(* IEC 61131-3 sources: AXOpen/src/showcase/app/src/core/AXOpen.Messaging, 3 files *)

(* ---- AxoIncidentBarExample.st ---- *)
USING AXOpen.Core;
USING AXOpen.Messaging;
USING AXOpen.Messaging.Static;

NAMESPACE AxoIncidentBarExample

    // Demonstrates AxoCauseAnalyzer + AxoIncidentBarView with a nested twin-tree topology.
    // Operator toggles condition BOOLs to fire Error/Critical messengers at multiple
    // tree levels. The bar ranks the upper messenger as 'top cause' because it
    // owns more downstream alarms (Symbol-prefix heuristic) and shares the burst window.
    {S7.extern=ReadWrite}
    CLASS IncidentTopology EXTENDS AXOpen.Core.AxoObject
        //<TopologyDeclaration>
        VAR PUBLIC
            {#ix-set:AttributeName = "<#Station (top of the topology)#>"}
            station : Station;
        END_VAR
        //</TopologyDeclaration>

        VAR PRIVATE
            _rootObject : AxoObject;
        END_VAR

        METHOD PUBLIC Execute
            _rootObject.Run(THIS);
            station.Run(_rootObject);
        END_METHOD
    END_CLASS

    {S7.extern=ReadWrite}
    CLASS PUBLIC Station EXTENDS AXOpen.Core.AxoObject
        //<StationDeclaration>
        VAR PUBLIC
            {#ix-set:AttributeName = "<#Station-level alarm (Error)#>"}
            {#ix-set:PlcTextList = "[1]:'<#Station emergency stop active#>':'<#Station has tripped the safety chain. Resolve all downstream issues before resetting.#>'"}
            _station_messenger : AXOpen.Messaging.Static.AxoMessenger;
            {#ix-set:AttributeName = "<#Trigger Station error#>"}
            _station_error : BOOL;

            {#ix-attr:[Container(Layout.Stack)]}
            drive : Drive;

            {#ix-attr:[Container(Layout.Stack)]}
            conveyor : Conveyor;
        END_VAR
        //</StationDeclaration>

        METHOD PUBLIC OVERRIDE Run
            VAR_INPUT
                inParent : IAxoObject;
            END_VAR
            SUPER.Run(inParent);
            _station_messenger.Serve(THIS);
            //<StationActivate>
            _station_messenger.ActivateOnCondition(ULINT#1, _station_error, eAxoMessageCategory#Error)
                              .RequireAcknowledgement();
            //</StationActivate>
            drive.Run(THIS);
            conveyor.Run(THIS);
        END_METHOD
    END_CLASS

    {S7.extern=ReadWrite}
    CLASS PUBLIC Drive EXTENDS AXOpen.Core.AxoObject
        //<DriveDeclaration>
        VAR PUBLIC
            {#ix-set:AttributeName = "<#Drive over-current (Critical)#>"}
            {#ix-set:PlcTextList = "[1]:'<#Drive over-current trip#>':'<#Inverter detected current above the safety limit. Check load and wiring.#>'"}
            _drive_messenger : AXOpen.Messaging.Static.AxoMessenger;
            {#ix-set:AttributeName = "<#Trigger Drive over-current#>"}
            _drive_error : BOOL;

            {#ix-attr:[Container(Layout.Stack)]}
            encoder : Encoder;
        END_VAR
        //</DriveDeclaration>

        METHOD PUBLIC OVERRIDE Run
            VAR_INPUT
                inParent : IAxoObject;
            END_VAR
            SUPER.Run(inParent);
            _drive_messenger.Serve(THIS);
            _drive_messenger.ActivateOnCondition(ULINT#1, _drive_error, eAxoMessageCategory#Critical)
                            .RequireAcknowledgement();
            encoder.Run(THIS);
        END_METHOD
    END_CLASS

    {S7.extern=ReadWrite}
    CLASS PUBLIC Encoder EXTENDS AXOpen.Core.AxoObject
        VAR PUBLIC
            {#ix-set:AttributeName = "<#Encoder signal lost (Error)#>"}
            {#ix-set:PlcTextList = "[1]:'<#Encoder signal lost#>':'<#The drive lost feedback from the encoder. Check cable continuity and connector seating.#>'"}
            _encoder_messenger : AXOpen.Messaging.Static.AxoMessenger;
            {#ix-set:AttributeName = "<#Trigger Encoder signal lost#>"}
            _encoder_error : BOOL;
        END_VAR

        METHOD PUBLIC OVERRIDE Run
            VAR_INPUT
                inParent : IAxoObject;
            END_VAR
            SUPER.Run(inParent);
            _encoder_messenger.Serve(THIS);
            _encoder_messenger.ActivateOnCondition(ULINT#1, _encoder_error, eAxoMessageCategory#Error)
                              .RequireAcknowledgement();
        END_METHOD
    END_CLASS

    {S7.extern=ReadWrite}
    CLASS PUBLIC Conveyor EXTENDS AXOpen.Core.AxoObject
        VAR PUBLIC
            {#ix-set:AttributeName = "<#Conveyor jammed (Error)#>"}
            {#ix-set:PlcTextList = "[1]:'<#Conveyor jammed#>':'<#Detected motor stall while pulley still commanded. Clear the obstruction and reset.#>'"}
            _conveyor_messenger : AXOpen.Messaging.Static.AxoMessenger;
            {#ix-set:AttributeName = "<#Trigger Conveyor jam#>"}
            _conveyor_error : BOOL;

            {#ix-attr:[Container(Layout.Stack)]}
            sensor : Sensor;
        END_VAR

        METHOD PUBLIC OVERRIDE Run
            VAR_INPUT
                inParent : IAxoObject;
            END_VAR
            SUPER.Run(inParent);
            _conveyor_messenger.Serve(THIS);
            _conveyor_messenger.ActivateOnCondition(ULINT#1, _conveyor_error, eAxoMessageCategory#Error)
                               .RequireAcknowledgement();
            sensor.Run(THIS);
        END_METHOD
    END_CLASS

    {S7.extern=ReadWrite}
    CLASS PUBLIC Sensor EXTENDS AXOpen.Core.AxoObject
        VAR PUBLIC
            {#ix-set:AttributeName = "<#Sensor disconnected (Error)#>"}
            {#ix-set:PlcTextList = "[1]:'<#Sensor disconnected#>':'<#Photo-eye lost present feedback. Verify alignment and 24V supply.#>'"}
            _sensor_messenger : AXOpen.Messaging.Static.AxoMessenger;
            {#ix-set:AttributeName = "<#Trigger Sensor disconnect#>"}
            _sensor_error : BOOL;
        END_VAR

        METHOD PUBLIC OVERRIDE Run
            VAR_INPUT
                inParent : IAxoObject;
            END_VAR
            SUPER.Run(inParent);
            _sensor_messenger.Serve(THIS);
            _sensor_messenger.ActivateOnCondition(ULINT#1, _sensor_error, eAxoMessageCategory#Error)
                             .RequireAcknowledgement();
        END_METHOD
    END_CLASS

END_NAMESPACE

(* ---- AxoStaticMessengerDocuExample.st ---- *)
USING AXOpen.Messaging;
USING AXOpen.Messaging.Static;

NAMESPACE AxoStaticMessengerDocuExample
    {S7.extern=ReadWrite}
    CLASS MessengersExamples EXTENDS AXOpen.Core.AxoObject
        VAR PUBLIC
            {#ix-set:AttributeName = "<#Messenger 1 - activate using 'Activate' method called inside the if statement#>"}
            {#ix-set:PlcTextList = "[1]:'<#Messenger 1: message text for message code 1#>':'<#Messenger 1: help text for message code 1#>';[2]:'<#Messenger 1: message text for message code 2#>':'<#Messenger 1: help text for message code 2#>';[3]:'<#Messenger 1: message text for message code 3#>':'<#Messenger 1: help text for message code 3#>';[4]:'<#Messenger 1: message text for message code 4#>':'<#Messenger 1: help text for message code 4#>';[5]:'<#Messenger 1: message text for message code 5#>':'<#Messenger 1: help text for message code 5#>';[6]:'<#Messenger 1: message text for message code 6#>':'<#Messenger 1: help text for message code 6#>';[7]:'<#Messenger 1: message text for message code 7#>':'<#Messenger 1: help text for message code 7#>';[8]:'<#Messenger 1: message text for message code 8#>':'<#Messenger 1: help text for message code 8#>';[9]:'<#Messenger 1: message text for message code 9#>':'<#Messenger 1: help text for message code 9#>';[10]:'<#Messenger 1: message text for message code 10#>':'<#Messenger 1: help text for message code 10#>';[11]:'<#Messenger 1: message text for message code 11#>':'<#Messenger 1: help text for message code 11#>'"}
            _messenger1 : AXOpen.Messaging.Static.AxoMessenger;
            {#ix-attr:[Container(Layout.Wrap)]}
            {#ix-set:AttributeName = "<#Set to high to activate the messenger 1#>"}
            _messenger1condition : BOOL;
            {#ix-set:AttributeName = "<#message 1 code#>"}
            _messenger1code : UINT;

            {#ix-attr:[Container(Layout.Stack)]}
            {#ix-set:AttributeName = "<#Messenger 2 - activate using 'ActivateOnCondition' method called cyclically#>"}
            {#ix-set:PlcTextList = "[1]:'<#Messenger 2: message text for message code 1#>':'<#Messenger 2: help text for message code 1#>'[2]:'<#Messenger 2: message text for message code 2#>':'<#Messenger 2: help text for message code 2#>'"}
            _messenger2 : AXOpen.Messaging.Static.AxoMessenger;
            {#ix-attr:[Container(Layout.Wrap)]}
            {#ix-set:AttributeName = "<#Set to high to activate the messenger 2#>"}
            _messenger2condition : BOOL;
            {#ix-set:AttributeName = "<#message 2 code#>"}
            _messenger2code : UINT;

            {#ix-attr:[Container(Layout.Stack)]}
            {#ix-set:AttributeName = "<#Messenger 3 - one message example, long help text#>"}
            {#ix-set:PlcTextList = "[1]:'<#Message text for messenger 3#>':'<#Lorem ipsum dolor sit amet, consectetur adipiscing elit. Phasellus neque eros, malesuada ac orci ut, ornare ullamcorper purus. Integer ultrices turpis vel est suscipit blandit. Mauris blandit eros augue, in mollis dui tincidunt vel. Sed placerat augue risus, eget pulvinar felis dictum quis. Aliquam ut interdum nisl. Aliquam et velit id turpis blandit laoreet nec ut ligula. Aliquam ac neque risus. Fusce porta mauris eget nulla iaculis mattis. Etiam auctor mi eget libero laoreet, sed interdum ipsum pellentesque. Maecenas vitae quam vitae velit tincidunt fringilla. Fusce sagittis elit sit amet tempor pretium. Donec elementum, ligula at laoreet mollis, est ipsum elementum lectus, et mollis nisi tellus id erat. In hac habitasse platea dictumst.#>'"}
            _messenger3 : AXOpen.Messaging.Static.AxoMessenger;
            {#ix-set:AttributeName = "<#Set to high to activate the messenger 3#>"}
            _messenger3condition : BOOL;

            {#ix-attr:[Container(Layout.Stack)]}
            //<PlcTextListDeclaration>
            {#ix-set:AttributeName = "<#Messenger 4 - textlist in PLC#>"}
            {#ix-set:PlcTextList = "[1]:'<#Messenger 4: static message text for message code 1 declared in the PLC code#>':'<#Messenger 4: static help text for message code 1 declared in the PLC code#>'[2]:'<#Messenger 4: static message text for message code 2 declared in the PLC code#>':'<#Messenger 4: static help text for message code 2 declared in the PLC code#>'"}
            _messenger4 : AXOpen.Messaging.Static.AxoMessenger;
            //</PlcTextListDeclaration>
            {#ix-set:AttributeName = "<#Set to high to activate the messenger 4 with message code 1#>"}
            _messenger4condition_1 : BOOL;
            {#ix-set:AttributeName = "<#Set to high to activate the messenger 4 with message code 2#>"}
            _messenger4condition_2 : BOOL;

            {#ix-attr:[Container(Layout.Stack)]}
            //<TextListGoingToBeDeclaredInDotNet>
            {#ix-set:AttributeName = "<#Messenger 5 - textlist in .NET#>"}
            _messenger5 : AXOpen.Messaging.Static.AxoMessenger;
            //</TextListGoingToBeDeclaredInDotNet>
            {#ix-attr:[Container(Layout.Wrap)]}
            {#ix-set:AttributeName = "<#Set to high to activate the messenger 5 with code 1#>"}
            _messenger5condition_1 : BOOL;
            {#ix-set:AttributeName = "<#Set to high to activate the messenger 5 with code 2#>"}
            _messenger5condition_2 : BOOL;
            {#ix-set:AttributeName = "<#Set to high to activate the messenger 5 with code 3#>"}
            _messenger5condition_3 : BOOL;
            {#ix-set:AttributeName = "<#Set to high to activate the messenger 5 with code 4#>"}
            _messenger5condition_4 : BOOL;
            {#ix-set:AttributeName = "<#Set to high to activate the messenger 5 with code 5#>"}
            _messenger5condition_5 : BOOL;
            {#ix-set:AttributeName = "<#Set to high to activate the messenger 5 with code 6#>"}
            _messenger5condition_6 : BOOL;
            {#ix-set:AttributeName = "<#Set to high to activate the messenger 5 with code 7#>"}
            _messenger5condition_7 : BOOL;
            {#ix-set:AttributeName = "<#Set to high to activate the messenger 5 with code 8#>"}
            _messenger5condition_8 : BOOL;
            {#ix-set:AttributeName = "<#Set to high to activate the messenger 5 with code 9#>"}
            _messenger5condition_9 : BOOL;
            {#ix-set:AttributeName = "<#Set to high to activate the messenger 5 with code 10, with no help text defined#>"}
            _messenger5condition_10 : BOOL;
            {#ix-set:AttributeName = "<#Set to high to call the messenger 5#>"}
            _messenger5callcondition : BOOL;

            {#ix-attr:[Container(Layout.Stack)]}
            {#ix-set:AttributeName = "<#Messenger 6 - invalid implementation#>"}
            {#ix-set:PlcTextList = "[1]:'<#Messenger 6: static message text for message code 1 declared in the PLC code#>':'<#Messenger 6: static help text for message code 1 declared in the PLC code#>'[2]:'<#Messenger 6: static message text for message code 2 declared in the PLC code#>':'<#Messenger 6: static help text for message code 2 declared in the PLC code#>'"}
            _messenger6 : AXOpen.Messaging.Static.AxoMessenger;
            {#ix-set:AttributeName = "<#Set to high to activate the messenger 6 with message code 1#>"}
            _messenger6condition_1 : BOOL;
            {#ix-set:AttributeName = "<#Set to high to activate the messenger 6 with message code 2#>"}
            _messenger6condition_2 : BOOL;
        END_VAR

        VAR PRIVATE
            _rootObject :   AxoObject;
        END_VAR
        METHOD PUBLIC Execute
            _rootObject.Run(THIS);
            //<Activate>
            _messenger1.Serve(_rootObject);
            IF _messenger1condition THEN
                _messenger1.Activate(_messenger1code,eAxoMessageCategory#Error);
            END_IF;
            //</Activate>

            //<ActivateOnCondition>
            _messenger2.Serve(_rootObject);
            _messenger2.ActivateOnCondition(_messenger2code,_messenger2condition,eAxoMessageCategory#Warning).RequireAcknowledgement();
            //</ActivateOnCondition>

            //<RequireAcknowledgement>
            _messenger2.Serve(_rootObject);
            _messenger2.ActivateOnCondition(_messenger2code,_messenger2condition,eAxoMessageCategory#Warning).RequireAcknowledgement();
            //</RequireAcknowledgement>

            //<DoNotRequireAcknowledgement>
            _messenger3.Serve(_rootObject);
            _messenger3.ActivateOnCondition(UINT#1,_messenger3condition,eAxoMessageCategory#Error).DoNotRequireAcknowledgement();
            //</DoNotRequireAcknowledgement>

            //<ActivateOnConditionWithMessageCodeTextListDeclaredInThePlcCode>
            _messenger4.Serve(_rootObject);
            _messenger4.ActivateOnCondition(UINT#1,_messenger4condition_1,eAxoMessageCategory#Info).RequireAcknowledgement();
            _messenger4.ActivateOnCondition(UINT#2,_messenger4condition_2,eAxoMessageCategory#Info).RequireAcknowledgement();
            //</ActivateOnConditionWithMessageCodeTextListDeclaredInThePlcCode>

            //<ActivateOnConditionWithMessageCodeTextListDeclaredInDotNet>
            IF _messenger5callcondition THEN
                _messenger5.Serve(_rootObject);
                _messenger5.ActivateOnCondition(ULINT#1,_messenger5condition_1,eAxoMessageCategory#Error).RequireAcknowledgement();
                _messenger5.ActivateOnCondition(ULINT#2,_messenger5condition_2,eAxoMessageCategory#Error).RequireAcknowledgement();
                _messenger5.ActivateOnCondition(ULINT#3,_messenger5condition_3,eAxoMessageCategory#Error).RequireAcknowledgement();
                _messenger5.ActivateOnCondition(ULINT#4,_messenger5condition_4,eAxoMessageCategory#Error).RequireAcknowledgement();
                _messenger5.ActivateOnCondition(ULINT#5,_messenger5condition_5,eAxoMessageCategory#Error).RequireAcknowledgement();
                _messenger5.ActivateOnCondition(ULINT#6,_messenger5condition_6,eAxoMessageCategory#Error).RequireAcknowledgement();
                _messenger5.ActivateOnCondition(ULINT#7,_messenger5condition_7,eAxoMessageCategory#Error).RequireAcknowledgement();
                _messenger5.ActivateOnCondition(ULINT#8,_messenger5condition_8,eAxoMessageCategory#Error).RequireAcknowledgement();
                _messenger5.ActivateOnCondition(ULINT#9,_messenger5condition_9,eAxoMessageCategory#Error).RequireAcknowledgement();
                _messenger5.ActivateOnCondition(ULINT#10,_messenger5condition_10,eAxoMessageCategory#Error).RequireAcknowledgement();
            ELSE
                _messenger5.Restore();
            END_IF;
            //</ActivateOnConditionWithMessageCodeTextListDeclaredInDotNet>

            //<InvalidImplementation>
            _messenger6.ActivateOnCondition(UINT#1,_messenger6condition_1,eAxoMessageCategory#Info).RequireAcknowledgement();
            _messenger6.ActivateOnCondition(UINT#2,_messenger6condition_2,eAxoMessageCategory#Info).RequireAcknowledgement();
            _messenger6.Serve(_rootObject);
            //</InvalidImplementation>
        END_METHOD
    END_CLASS

    //<MessengerCompleteExample
    {S7.extern=ReadWrite}
    CLASS Messengers EXTENDS AXOpen.Core.AxoObject
        VAR PUBLIC
            {#ix-set:PlcTextList = "[10]:'<#Messenger 1: static message text for message code 10 declared in the PLC code#>':'<#Messenger 1: static help text for message code 10 declared in the PLC code#>'"}
            _messenger1 : AXOpen.Messaging.Static.AxoMessenger;
            {#ix-set:AttributeName = "<#Set to high to activate the messenger 1#>"}
            _messenger1condition : BOOL;

            {#ix-set:PlcTextList = "[10]:'<#Messenger 2: static message text for message code 10 declared in the PLC code#>':'<#Messenger 2: static help text for message code 10 declared in the PLC code#>'"}
            _messenger2 : AXOpen.Messaging.Static.AxoMessenger;
            {#ix-set:AttributeName = "<#Set to high to activate the messenger 2#>"}
            _messenger2condition : BOOL;

            {#ix-set:PlcTextList = "[10]:'<#Messenger 3: static message text for message code 10 declared in the PLC code#>':'<#Messenger 3: static help text for message code 10 declared in the PLC code#>';[20]:'<#Messenger 3: static message text for message code 20 declared in the PLC code#>':'<#Messenger 3: static help text for message code 20 declared in the PLC code#>'"}
            _messenger3 : AXOpen.Messaging.Static.AxoMessenger;
            {#ix-set:AttributeName = "<#Set to high to activate the messenger 3 with message code 10#>"}
            _messenger3condition_10 : BOOL;
            {#ix-set:AttributeName = "<#Set to high to activate the messenger 3 with message code 20#>"}
            _messenger3condition_20 : BOOL;

            _messenger4 : AXOpen.Messaging.Static.AxoMessenger;
            {#ix-set:AttributeName = "<#Set to high to activate the messenger 4 with message code 10#>"}
            _messenger4condition_10 : BOOL;
            {#ix-set:AttributeName = "<#Set to high to activate the messenger 4 with message code 20#>"}
            _messenger4condition_20 : BOOL;
        END_VAR
        VAR PRIVATE
            _rootObject :   AxoObject;
        END_VAR
        METHOD PUBLIC Execute
            _rootObject.Run(THIS);
            _messenger1.Serve(_rootObject);
            IF _messenger1condition THEN
                _messenger1.Activate(ULINT#10,eAxoMessageCategory#Error);
            END_IF;

            _messenger2.Serve(_rootObject);
            _messenger2.ActivateOnCondition(ULINT#10,_messenger2condition,eAxoMessageCategory#Warning);

            _messenger3.Serve(_rootObject);
            _messenger3.ActivateOnCondition(ULINT#10,_messenger3condition_10,eAxoMessageCategory#Error).DoNotRequireAcknowledgement();
            _messenger3.ActivateOnCondition(ULINT#20,_messenger3condition_20,eAxoMessageCategory#Warning).RequireAcknowledgement();

            _messenger4.Serve(_rootObject);
            _messenger4.ActivateOnCondition(ULINT#10,_messenger4condition_10,eAxoMessageCategory#Warning);
            _messenger4.ActivateOnCondition(ULINT#20,_messenger4condition_20,eAxoMessageCategory#Warning);

        END_METHOD
    END_CLASS
    //</MessengerCompleteExample
END_NAMESPACE

(* ---- AxoStaticMessengerExample.st ---- *)
USING AXOpen.Core;
USING AXOpen.Messaging;
USING AXOpen.Messaging.Static;

NAMESPACE AxoStaticMessengerExample

    {S7.extern=ReadWrite}
    CLASS Messengers EXTENDS AXOpen.Core.AxoObject
        VAR PUBLIC
            {#ix-set:AttributeName = "<#Messenger 1 - activate using 'Activate' method called inside the if statement#>"}
            {#ix-set:PlcTextList = "[1]:'<#Messenger 1: message text for message code 1#>':'<#Messenger 1: help text for message code 1#>';[2]:'<#Messenger 1: message text for message code 2#>':'<#Messenger 1: help text for message code 2#>';[3]:'<#Messenger 1: message text for message code 3#>':'<#Messenger 1: help text for message code 3#>';[4]:'<#Messenger 1: message text for message code 4#>':'<#Messenger 1: help text for message code 4#>';[5]:'<#Messenger 1: message text for message code 5#>':'<#Messenger 1: help text for message code 5#>';[6]:'<#Messenger 1: message text for message code 6#>':'<#Messenger 1: help text for message code 6#>';[7]:'<#Messenger 1: message text for message code 7#>':'<#Messenger 1: help text for message code 7#>';[8]:'<#Messenger 1: message text for message code 8#>':'<#Messenger 1: help text for message code 8#>';[9]:'<#Messenger 1: message text for message code 9#>':'<#Messenger 1: help text for message code 9#>';[10]:'<#Messenger 1: message text for message code 10#>':'<#Messenger 1: help text for message code 10#>';[11]:'<#Messenger 1: message text for message code 11#>':'<#Messenger 1: help text for message code 11#>'"}
            _messenger1 : AXOpen.Messaging.Static.AxoMessenger;
            {#ix-attr:[Container(Layout.Wrap)]}
            {#ix-set:AttributeName = "<#Set to high to activate the messenger 1#>"}
            _messenger1condition : BOOL;
            {#ix-set:AttributeName = "<#message 1 code#>"}
            _messenger1code : UINT;

            {#ix-attr:[Container(Layout.Stack)]}
            {#ix-set:AttributeName = "<#Messenger 2 - activate using 'ActivateOnCondition' method called cyclically#>"}
            {#ix-set:PlcTextList = "[1]:'<#Messenger 2: message text for message code 1#>':'<#Messenger 2: help text for message code 1#>'[2]:'<#Messenger 2: message text for message code 2#>':'<#Messenger 2: help text for message code 2#>'"}
            _messenger2 : AXOpen.Messaging.Static.AxoMessenger;
            {#ix-attr:[Container(Layout.Wrap)]}
            {#ix-set:AttributeName = "<#Set to high to activate the messenger 2#>"}
            _messenger2condition : BOOL;
            {#ix-set:AttributeName = "<#message 2 code#>"}
            _messenger2code : UINT;

            {#ix-attr:[Container(Layout.Stack)]}
            {#ix-set:AttributeName = "<#Messenger 3 - one message example, long help text#>"}
            {#ix-set:PlcTextList = "[1]:'<#Message text for messenger 3#>':'<#Lorem ipsum dolor sit amet, consectetur adipiscing elit. Phasellus neque eros, malesuada ac orci ut, ornare ullamcorper purus. Integer ultrices turpis vel est suscipit blandit. Mauris blandit eros augue, in mollis dui tincidunt vel. Sed placerat augue risus, eget pulvinar felis dictum quis. Aliquam ut interdum nisl. Aliquam et velit id turpis blandit laoreet nec ut ligula. Aliquam ac neque risus. Fusce porta mauris eget nulla iaculis mattis. Etiam auctor mi eget libero laoreet, sed interdum ipsum pellentesque. Maecenas vitae quam vitae velit tincidunt fringilla. Fusce sagittis elit sit amet tempor pretium. Donec elementum, ligula at laoreet mollis, est ipsum elementum lectus, et mollis nisi tellus id erat. In hac habitasse platea dictumst.#>'"}
            _messenger3 : AXOpen.Messaging.Static.AxoMessenger;
            {#ix-set:AttributeName = "<#Set to high to activate the messenger 3#>"}
            _messenger3condition : BOOL;

            {#ix-attr:[Container(Layout.Stack)]}
            {#ix-set:AttributeName = "<#Messenger 4 - textlist in PLC#>"}
            {#ix-set:PlcTextList = "[1]:'<#Messenger 4: static message text for message code 1 declared in the PLC code#>':'<#Messenger 4: static help text for message code 1 declared in the PLC code#>'[2]:'<#Messenger 4: static message text for message code 2 declared in the PLC code#>':'<#Messenger 4: static help text for message code 2 declared in the PLC code#>'"}
            _messenger4 : AXOpen.Messaging.Static.AxoMessenger;
            {#ix-set:AttributeName = "<#Set to high to activate the messenger 4 with message code 1#>"}
            _messenger4condition_1 : BOOL;
            {#ix-set:AttributeName = "<#Set to high to activate the messenger 4 with message code 2#>"}
            _messenger4condition_2 : BOOL;
            {#ix-set:AttributeName = "<#Message to be posted by messenger 4 #>"}
            _messenger4text : STRING[254] := 'Messenger 4 text';
            {#ix-set:AttributeName = "<#Set to high to post dynamic message to messanger 4#>"}
            _messenger4condition_3 : BOOL;

            {#ix-attr:[Container(Layout.Stack)]}
            {#ix-set:AttributeName = "<#Messenger 5 - textlist in .NET#>"}
            _messenger5 : AXOpen.Messaging.Static.AxoMessenger;
            {#ix-attr:[Container(Layout.Wrap)]}
            {#ix-set:AttributeName = "<#Set to high to activate the messenger 5 with code 1#>"}
            _messenger5condition_1 : BOOL;
            {#ix-set:AttributeName = "<#Set to high to activate the messenger 5 with code 2#>"}
            _messenger5condition_2 : BOOL;
            {#ix-set:AttributeName = "<#Set to high to activate the messenger 5 with code 3#>"}
            _messenger5condition_3 : BOOL;
            {#ix-set:AttributeName = "<#Set to high to activate the messenger 5 with code 4#>"}
            _messenger5condition_4 : BOOL;
            {#ix-set:AttributeName = "<#Set to high to activate the messenger 5 with code 5#>"}
            _messenger5condition_5 : BOOL;
            {#ix-set:AttributeName = "<#Set to high to activate the messenger 5 with code 6#>"}
            _messenger5condition_6 : BOOL;
            {#ix-set:AttributeName = "<#Set to high to activate the messenger 5 with code 7#>"}
            _messenger5condition_7 : BOOL;
            {#ix-set:AttributeName = "<#Set to high to activate the messenger 5 with code 8#>"}
            _messenger5condition_8 : BOOL;
            {#ix-set:AttributeName = "<#Set to high to activate the messenger 5 with code 9#>"}
            _messenger5condition_9 : BOOL;
            {#ix-set:AttributeName = "<#Set to high to activate the messenger 5 with code 10, with no help text defined#>"}
            _messenger5condition_10 : BOOL;
            {#ix-set:AttributeName = "<#Message to be posted by messenger 5#>"}
            _messenger5text : STRING[254] := 'Messenger 5 text';
            {#ix-set:AttributeName = "<#Set to high to post dynamic message to messanger 5#>"}
            _messenger5condition_11 : BOOL;

            {#ix-set:AttributeName = "<#Set to high to call the messenger 5#>"}
            _messenger5callcondition : BOOL;

            {#ix-attr:[Container(Layout.Stack)]}
            {#ix-set:AttributeName = "<#Messenger 6 - invalid implementation#>"}
            {#ix-set:PlcTextList = "[1]:'<#Messenger 6: static message text for message code 1 declared in the PLC code#>':'<#Messenger 6: static help text for message code 1 declared in the PLC code#>'[2]:'<#Messenger 6: static message text for message code 2 declared in the PLC code#>':'<#Messenger 6: static help text for message code 2 declared in the PLC code#>'"}
            _messenger6 : AXOpen.Messaging.Static.AxoMessenger;
            {#ix-set:AttributeName = "<#Set to high to activate the messenger 6 with message code 1#>"}
            _messenger6condition_1 : BOOL;
            {#ix-set:AttributeName = "<#Set to high to activate the messenger 6 with message code 2#>"}
            _messenger6condition_2 : BOOL;
        END_VAR
        VAR PRIVATE
            _rootObject :   AxoObject;
        END_VAR
        METHOD PUBLIC Execute
            _rootObject.Run(THIS);

            _messenger1.Serve(_rootObject);
            IF _messenger1condition THEN
                _messenger1.Activate(_messenger1code,eAxoMessageCategory#Error);
            END_IF;

            _messenger2.Serve(_rootObject);
            _messenger2.ActivateOnCondition(_messenger2code,_messenger2condition,eAxoMessageCategory#Warning).RequireAcknowledgement();

            _messenger3.Serve(_rootObject);
            _messenger3.ActivateOnCondition(UINT#1,_messenger3condition,eAxoMessageCategory#Error).DoNotRequireAcknowledgement();

            _messenger4.Serve(_rootObject);
            _messenger4.ActivateOnCondition(UINT#1,_messenger4condition_1,eAxoMessageCategory#Info).RequireAcknowledgement();
            _messenger4.ActivateOnCondition(UINT#2,_messenger4condition_2,eAxoMessageCategory#Info).RequireAcknowledgement();

            IF _messenger4condition_3 THEN
                _messenger4.Post(inParent := _rootObject, inMessage := _messenger4text, inCategory := eAxoMessageCategory#Info) ;
            END_IF;

            IF _messenger5callcondition THEN
                _messenger5.Serve(_rootObject);
                _messenger5.ActivateOnCondition(ULINT#1,_messenger5condition_1,eAxoMessageCategory#Error).RequireAcknowledgement();
                _messenger5.ActivateOnCondition(ULINT#2,_messenger5condition_2,eAxoMessageCategory#Error).RequireAcknowledgement();
                _messenger5.ActivateOnCondition(ULINT#3,_messenger5condition_3,eAxoMessageCategory#Error).RequireAcknowledgement();
                _messenger5.ActivateOnCondition(ULINT#4,_messenger5condition_4,eAxoMessageCategory#Error).RequireAcknowledgement();
                _messenger5.ActivateOnCondition(ULINT#5,_messenger5condition_5,eAxoMessageCategory#Error).RequireAcknowledgement();
                _messenger5.ActivateOnCondition(ULINT#6,_messenger5condition_6,eAxoMessageCategory#Error).RequireAcknowledgement();
                _messenger5.ActivateOnCondition(ULINT#7,_messenger5condition_7,eAxoMessageCategory#Error).RequireAcknowledgement();
                _messenger5.ActivateOnCondition(ULINT#8,_messenger5condition_8,eAxoMessageCategory#Error).RequireAcknowledgement();
                _messenger5.ActivateOnCondition(ULINT#9,_messenger5condition_9,eAxoMessageCategory#Error).RequireAcknowledgement();
                _messenger5.ActivateOnCondition(ULINT#10,_messenger5condition_10,eAxoMessageCategory#Error).RequireAcknowledgement();
                IF _messenger5condition_11 THEN
                    _messenger5.Post(inParent := _rootObject, inMessage := _messenger5text, inCategory := eAxoMessageCategory#Info).RequireAcknowledgement();
                END_IF;
            ELSE
                _messenger5.Restore();
            END_IF;

            _messenger6.ActivateOnCondition(UINT#1,_messenger6condition_1,eAxoMessageCategory#Info).RequireAcknowledgement();
            _messenger6.ActivateOnCondition(UINT#2,_messenger6condition_2,eAxoMessageCategory#Info).RequireAcknowledgement();
            _messenger6.Serve(_rootObject);

        END_METHOD
    END_CLASS
END_NAMESPACE
